Staubli VAL3: readCNV.pgx

program readCNV(num& x_nError[] (dimensions=1))
  local bool l_bQuit
  local num l_nError
  local num l_nStep
  local string l_sValue
begin
  // This program initializes the parameters of the conveyor library
  // to be displayed in the Setting page of the user interface.
  //
  //   - Initializes List object fields (e.g. Encoder library)
  //----------------------------------------------------------------
  //
  x_nError=0
  l_nStep=0
  // Read current value from conveyor library
  resize(sCaption,1,pg:nNumOfTxtBox)
  call pg:getCaption(sCaption)
  //
  l_bQuit=false
  do
    switch l_nStep
      //*** FIELD ENCODER LIBRARY
      case 0
        // Initialize the List object
        resize(sItemList,1,1)
        if libList(cfg:sPATHENCODER,sItemList)==true
          call pg:setListOfItems(0,sItemList,l_nError)
        endIf
        if l_nError!=0
          l_bQuit=true
          x_nError=l_nError
        else
          // Read name of associated Encoder library
          l_sValue=cnv:sEncoderLib
          call pg:setFieldValue(sCaption[0],l_sValue,l_nError)
          l_nStep=10
        endIf
      break
      //*** FIELD DETECTION LIBRARY
      case 10
        //Initialize the List object
        resize(sItemList,1,1)
        if libList(cfg:sPATHDETECTION,sItemList)==true
          call pg:setListOfItems(1,sItemList,l_nError)
        endIf
        if l_nError!=0
          l_bQuit=true
          x_nError=l_nError
        else
          // Read name of associated Detection library
          l_sValue=cnv:sDetectionLib
          call pg:setFieldValue(sCaption[1],l_sValue,l_nError)
          l_nStep=20
        endIf
      break
      //*** FIELD CLOCK SIGNAL
      case 20
        //Initialize the List object
        call pg:setListOfItems(8,sDOutputsList,l_nError)
        if l_nError!=0
          l_bQuit=true
          x_nError=l_nError
        else
          //Force value
          l_sValue=cnv:sClockSigName
          call pg:setFieldValue(sCaption[8],l_sValue,l_nError)
          l_nStep=30
        endIf
      break
      //*** FIELD ThruUpLim
      case 30
        //Initialize the List object
        call pg:setListOfItems(5,sDOutputsList,l_nError)
        if l_nError!=0
          l_bQuit=true
          x_nError=l_nError
        else
          //Force value
          l_sValue=cnv:sUpLimSigName
          call pg:setFieldValue(sCaption[5],l_sValue,l_nError)
          l_nStep=40
        endIf
      break
      //*** FIELD ThruDwnLim
      case 40
        //Initialize the List object
        call pg:setListOfItems(6,sDOutputsList,l_nError)
        if l_nError!=0
          l_bQuit=true
          x_nError=l_nError
        else
          //Force value
          l_sValue=cnv:sDwnLimSigName
          call pg:setFieldValue(sCaption[6],l_sValue,l_nError)
          l_nStep=50
        endIf
      break
      //*** FIELD Event logging
      case 50
        if cnv:bLOG
          l_sValue="TRUE"
        else
          l_sValue="FALSE"
        endIf
        call pg:setFieldValue(sCaption[11],l_sValue,l_nError)
        l_nStep=60
      break
      // FURTHER FIELDS OF THE PAGE
      case 60
        // Height of the tracking window
        call ut:_toString(cnv:nTrackWinHeight,"",l_sValue)
        call pg:setFieldValue(sCaption[4],l_sValue,l_nError)
        // Size of the queue
        call ut:_toString(cnv:nBufferSize,"",l_sValue)
        call pg:setFieldValue(sCaption[2],l_sValue,l_nError)
        // Display ScaleFactor
        call ut:_toString(cnv:nENCSCALEFACTOR,".7",l_sValue)
        call pg:setFieldValue(sCaption[3],l_sValue,l_nError)
        // Detection matching tolerance
        call ut:_toString(cnv:nPosMatchTol,"",l_sValue)
        call pg:setFieldValue(sCaption[7],l_sValue,l_nError)
        // Clock period
        call ut:_toString(cnv:nClockPeriod,"",l_sValue)
        call pg:setFieldValue(sCaption[9],l_sValue,l_nError)
        // latch lock distance
        call ut:_toString(cnv:nLatchLockDist,"",l_sValue)
        call pg:setFieldValue(sCaption[10],l_sValue,l_nError)
        //
        l_bQuit=true
      break
    endSwitch
  until l_bQuit
end
